FUNCTION_BLOCK Machine EXTENDS PML_Method_Base
VAR
	XtsModuleRunner : ObjectRunner;
	xtsStateMachine : PMLStateMachine;
	Movers : ARRAY[0..7] OF XtsMover;
	iMovers : ARRAY[0..7] OF I_XtsMover := [Movers[0],Movers[1],
											Movers[2],Movers[3],
											Movers[4],Movers[5],
											Movers[6],Movers[7]];
	Station1 : StationSample := (Position := 850.0, 
									TempPropTime := T#1500MS);
	Station2 : StationSample := (Position := 1200.0, 
									TempPropTime := T#1500MS);
	Station3 : StationSample := (Position := 1450.0, 
									TempPropTime := T#500MS);
	Station4 : StationSample := (Position := 2100.0, 
									TempPropTime := T#1500MS);
	Station5 : StationSample := (Position := 2400.0, 
									TempPropTime := T#1500MS);
	iStationArray : ARRAY[0..SystemParameters.NumberOfStations] OF IProcess := [Station1,Station2,
																					Station3,Station4,
																					Station5];//,Station6];
	systemXtsioEnvVar : XtsIoEnvVar;	
	systemXtsHardware : XTSHardware;				
	systemCAGroup : CollisionGroup;															
	MyXts : ThisXTS(systemXtsioEnvVar,systemXtsHardware,systemCAGroup) := (MyXts := 1, ExpectedNumberOfParts := 1, ExpectedNumberOfTracks := 1);
	MoverSequences : ARRAY[0..7] OF IndexMoverSequence := [8((MyStations := iStationArray,
																				MyStartPosition := 1000.0))];	
	i : INT;
	RegisterationComplete : BOOL;
	Mover1ActiveTrack: INT;
END_VAR
VAR CONSTANT
	NumberOFSystemMovers : INT := 8;
END_VAR

METHOD PROTECTED Aborting : BOOL
VAR_INPUT
END_VAR
IF MyXts.DisableXTS() THEN
	ipackml.SetStateComplete();
END_IF
END_METHOD

METHOD PROTECTED Clearing : BOOL
VAR_INPUT
END_VAR
MyXts.ActivateTracksInMovers();
ipackml.SetStateComplete();
END_METHOD

METHOD Cycle : HRESULT
SUPER^.Cycle();
xtsStateMachine.Cycle();
XtsModuleRunner.Cycle();
END_METHOD

METHOD GetPackML : E_PMLState;
VAR_INPUT
END_VAR
GetPackML := xtsStateMachine.GetCurrentState();
END_METHOD

METHOD Initialise : BOOL
VAR_INPUT
END_VAR
IF NOT RegisterationComplete THEN
	FOR i := 0 TO 7 DO
		XtsModuleRunner.RegisterModule(Movers[i]);
		XtsModuleRunner.RegisterModule(MoverSequences[i]);
		MoverSequences[i].MyMover := Movers[i]; 
	END_FOR
	XtsModuleRunner.RegisterModule(systemXtsioEnvVar);
	XtsModuleRunner.RegisterModule(systemXtsHardware);
	XtsModuleRunner.RegisterModule(systemCAGroup);
	XtsModuleRunner.RegisterModule(MyXts);
	XtsModuleRunner.RegisterModule(Station1);
	XtsModuleRunner.RegisterModule(Station2);
	XtsModuleRunner.RegisterModule(Station3);
	XtsModuleRunner.RegisterModule(Station4);
	XtsModuleRunner.RegisterModule(Station5);
	THIS^.PackMLStateMachine := xtsStateMachine;
	xtsStateMachine.PmlModeCommand(Mode := E_PMLProtectedUnitMode.ePMLProtUnitMode_Production);
	xtsStateMachine.PmlStateCommand(Command := E_PMLCommand.ePMLCommand_Abort);
	RegisterationComplete := TRUE;
END_IF

IF XtsModuleRunner.Initialise() = 1 THEN
	Initialise := TRUE;
	FOR i := 0 TO 7 DO
		MyXts.RegisterMovers(MyMover := iMovers[i]);
	END_FOR
END_IF
END_METHOD

METHOD PROTECTED Resetting : BOOL
VAR_INPUT
END_VAR
IF NOT MyXts.IsXtsReady() THEN
	MyXts.EnableXTS();
ELSE
	ipackml.SetStateComplete();
END_IF
END_METHOD

{attribute 'TcRpcEnable':='1'}
METHOD SetPackML : BOOL
VAR_INPUT
	state : E_PMLCommand;
END_VAR
xtsStateMachine.PmlStateCommand(Command := state);
END_METHOD

METHOD PROTECTED Starting : BOOL
VAR_INPUT
END_VAR
MyXts.MoverHomeSequence();
ipackml.SetStateComplete();
Mover1ActiveTrack := iMovers[0].MoversActiveTrack;
END_METHOD

END_FUNCTION_BLOCK

(* stored: Version 1.1.0.1, ProductVersion 3.1.4026.12
   POU Machine: Id {e8d4edde-6e68-4e80-9f5b-2e9346044142}, SpecialFunc None
   Method Aborting: Id {5e47e9ec-af05-4f55-a014-ec50066f7440}
   Method Clearing: Id {29611cf3-b33d-4081-8744-6b6cb57a9ba1}
   Method Cycle: Id {800ade8f-bb7c-4681-a005-35c2c0ff3879}
   Method GetPackML: Id {f4fa13f0-e9c7-4904-acb1-6e313a496be6}
   Method Initialise: Id {4069299b-b0bd-441e-b636-7c39202b14ad}
   Method Resetting: Id {9f1f9d34-e777-4487-9353-8daf70debb65}
   Method SetPackML: Id {53c56351-61ed-4063-8940-94e0a76b1fed}
   Method Starting: Id {6289f1df-c8c2-4a24-9238-0ac10992d955} *)
